PROGRAM P_Demo_UInt64Div64Ex
VAR
    uliNanos   : T_ULARGE_INTEGER;; // 累计纳秒
    uliDivisor : T_ULARGE_INTEGER;; // 1e9 = 一秒的纳秒数
    uliSeconds : T_ULARGE_INTEGER;; // 秒数（商）
    uliSubNs   : T_ULARGE_INTEGER;; // 亚秒纳秒（余数）
    bCompute   : BOOL;
END_VAR

// ============================================================
// Tc2_Utilities.UInt64Div64Ex 演示程序（FUNCTION，单周期触发）
// ============================================================
// 场景：把累计纳秒数同时拆成秒数（商）+ 纳秒余数（亚秒部分）用于显示。
// 价值：一次硬件除法同时拿商与余数，比两次调用快一倍。
// 验证步骤：
//   1. 把本 PROGRAM 加到 PlcTask 调用列表
//   2. 编译 + 登录
//   3. 在线把 b... 触发位置 TRUE 一个周期
//   4. 观察输出变量是否符合期望
// ============================================================

uliDivisor := ULARGE_INTEGER(0, 1000000000);   // 1e9
IF bCompute AND NOT UInt64isZero(uliDivisor) THEN
    uliSeconds := UInt64Div64Ex(uliNanos, uliDivisor, uliSubNs);
    bCompute := FALSE;
END_IF;

END_PROGRAM

(* stored: Version 1.1.0.1, ProductVersion 3.1.4024.5
   POU P_Demo_UInt64Div64Ex: Id {41900e72-c1d9-597c-8230-192215dd3fc5}, SpecialFunc None *)
